{attribute addProperty BoxType "EM3701-0000-0016"}
{attribute addProperty Id "AI_InputsAT %I*AI_Inputs_D7666BC23240WcStateAT %I*WcState_98A4DF7520.250InfoDataAT %I*InfoData_BC63D37F80100"}
{attribute addProperty CRC "372664775"}
{attribute addProperty SizeInBites "114"}
{attribute addProperty SizeInBytes "14.25"}
TYPE EM3701_6ABA943A :
STRUCT
	{attribute addProperty Name "AI_Inputs"}
	AI_Inputs : AI_Inputs_D7666BC2;
	{attribute addProperty Name "WcState"}
	WcState : WcState_98A4DF75;
	{attribute addProperty Name "InfoData"}
	InfoData : InfoData_BC63D37F;
END_STRUCT
END_TYPE

(* stored: Version 1.2.0.0, ProductVersion 3.1.4024.9
   DUT EM3701_6ABA943A: Id {28ff33af-e2e6-4309-b79b-a0683c57f74a} *)
